GLOBALCONSTANTS AID_SK (* Soft key object attribute ids *)
  (* Standard: 61499-1; Description: Copyright (c) 2023 HR Agrartechnik GmbH This program and the accompanying materials are made available under the terms of the Eclipse Public License 2.0 which is available at https://www.eclipse.org/legal/epl-2.0/ SPDX-License-Identifier: EPL-2.0 *)
  (* Version 1.0, 2026-06-20, Franz Höpfinger, HR Agrartechnik GmbH *)
  PACKAGE isobus::UT::Q::const::AID;
  VAR_GLOBAL CONSTANT
    BACKGROUND_COLOUR : USINT := USINT#1; (* 1: AID_SK_BACKGROUND_COLOUR - Background colour index. *)
    KEY_CODE : USINT := USINT#2; (* 2: AID_SK_KEY_CODE - [2] Read-only attribute. VT reports this code in the Soft Key Activation message. *)
  END_VAR
END_GLOBALCONSTANTS
